// Mitsubishi GX Works2 project: zadatak_1_with_error   PLC: FX3S

// global labels: Global1
VAR_GLOBAL
  out_zone : zona_izlaza;
  fsm_1 : fsm;
  in_zone : zona_ulaza;
END_VAR

// task Task_01 (event TRUE, interval 0, priority 31): POU_01

PROGRAM POU_01
VAR
  system_on : BOOL;
  start : BOOL;
  stop_all : BOOL;
  start_all : BOOL;
  pump_on : BOOL;
  goto_1 : BOOL;
  goto_2 : BOOL;
  goto_3 : BOOL;
  goto_4 : BOOL;
  goto_0 : BOOL;
  cur_state : INT;
  s_0 : BOOL;
  s_1 : BOOL;
  s_2 : BOOL;
  s_3 : BOOL;
  s_4 : BOOL;
  sensor_2 : BOOL;
END_VAR
VAR CONSTANT
  pause : TIME := T#10s;
END_VAR
VAR
  elapsed_time : TIME;
  sensor_1 : BOOL;
  water_rising : BOOL;
  valve_1 : BOOL;
  motor : BOOL;
  water_falling : BOOL;
  valve_2 : BOOL;
  alarm : BOOL;
  TON_1 : TON;
  cnt_cycles_1 : cnt_cycles;
  done : BOOL;
  blink_1 : blink;
  lamp : BOOL;
  state : INT;
  enb : BOOL;
  sON : BOOL;
  zona_izlaz : zona_izlaza;
  zona_ulazz : zona_ulaza;
END_VAR
(* structured ladder/FBD written out as ST: instructions are called as NAME(EN, inputs, outputs); _pN, _eN, _tN stand for wires *)
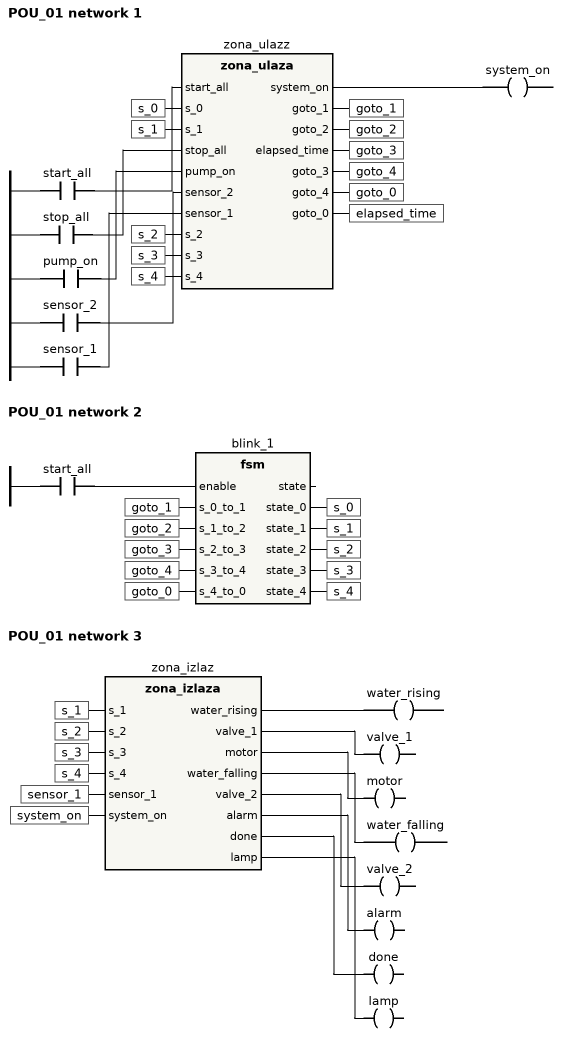
(* network 1 *)
zona_ulazz(start_all := start_all, s_0 := s_0, s_1 := s_1, stop_all := stop_all, pump_on := pump_on, sensor_2 := sensor_2, sensor_1 := sensor_1, s_2 := s_2, s_3 := s_3, s_4 := s_4, goto_1 => goto_1, goto_2 => goto_2, elapsed_time => goto_3, goto_3 => goto_4, goto_4 => goto_0, goto_0 => elapsed_time);
system_on := zona_ulazz.system_on;
(* network 2 *)
blink_1(enable := start_all, s_0_to_1 := goto_1, s_1_to_2 := goto_2, s_2_to_3 := goto_3, s_3_to_4 := goto_4, s_4_to_0 := goto_0, state_0 => s_0, state_1 => s_1, state_2 => s_2, state_3 => s_3, state_4 => s_4);
(* network 3 *)
zona_izlaz(s_1 := s_1, s_2 := s_2, s_3 := s_3, s_4 := s_4, sensor_1 := sensor_1, system_on := system_on);
water_rising := zona_izlaz.water_rising;
valve_1 := zona_izlaz.valve_1;
motor := zona_izlaz.motor;
water_falling := zona_izlaz.water_falling;
valve_2 := zona_izlaz.valve_2;
alarm := zona_izlaz.alarm;
done := zona_izlaz.done;
lamp := zona_izlaz.lamp;
END_PROGRAM

FUNCTION_BLOCK fsm
VAR_OUTPUT
  state : INT;
END_VAR
VAR CONSTANT
  cmp_with_0 : INT;
END_VAR
VAR
  is_eqv : ARRAY [0..2] OF BOOL;
END_VAR
VAR_INPUT
  enable : BOOL;
  s_0_to_1 : BOOL;
END_VAR
VAR_OUTPUT
  state_0 : BOOL;
END_VAR
VAR CONSTANT
  cmp_with_1 : INT := 1;
END_VAR
VAR_INPUT
  s_1_to_2 : BOOL;
END_VAR
VAR_OUTPUT
  state_1 : BOOL;
END_VAR
VAR CONSTANT
  cmp_with_2 : INT := 2;
END_VAR
VAR_INPUT
  s_2_to_3 : BOOL;
END_VAR
VAR_OUTPUT
  state_2 : BOOL;
  state_3 : BOOL;
END_VAR
VAR_INPUT
  s_3_to_4 : BOOL;
END_VAR
VAR CONSTANT
  cmp_with_4 : INT := 4;
  cmp_with_3 : INT := 3;
END_VAR
VAR_OUTPUT
  state_4 : BOOL;
END_VAR
VAR_INPUT
  s_4_to_0 : BOOL;
END_VAR
VAR
  blink_1 : blink;
END_VAR
(* structured ladder/FBD written out as ST: instructions are called as NAME(EN, inputs, outputs); _pN, _eN, _tN stand for wires *)
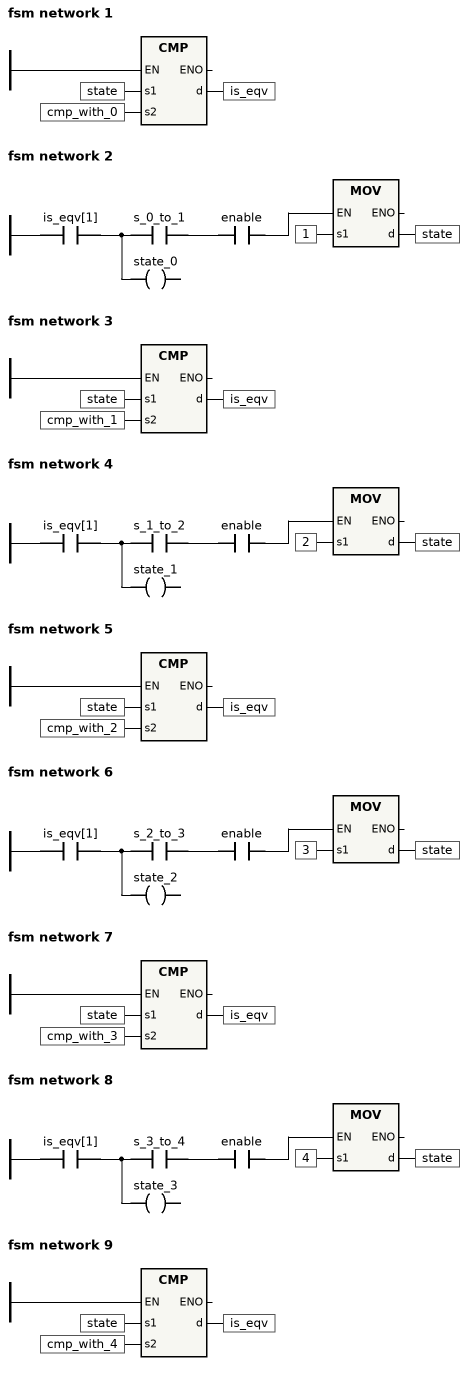
(* network 1 *)
CMP(TRUE, state, cmp_with_0, is_eqv);
(* network 2 *)
MOV(is_eqv[1] AND s_0_to_1 AND enable, 1, state);
state_0 := is_eqv[1];
(* network 3 *)
CMP(TRUE, state, cmp_with_1, is_eqv);
(* network 4 *)
MOV(is_eqv[1] AND s_1_to_2 AND enable, 2, state);
state_1 := is_eqv[1];
(* network 5 *)
CMP(TRUE, state, cmp_with_2, is_eqv);
(* network 6 *)
MOV(is_eqv[1] AND s_2_to_3 AND enable, 3, state);
state_2 := is_eqv[1];
(* network 7 *)
CMP(TRUE, state, cmp_with_3, is_eqv);
(* network 8 *)
MOV(is_eqv[1] AND s_3_to_4 AND enable, 4, state);
state_3 := is_eqv[1];
(* network 9 *)
CMP(TRUE, state, cmp_with_4, is_eqv);
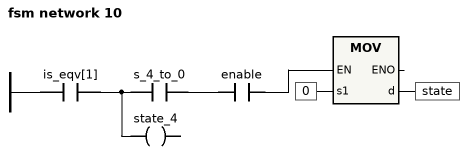
(* network 10 *)
MOV(is_eqv[1] AND s_4_to_0 AND enable, 0, state);
state_4 := is_eqv[1];
END_FUNCTION_BLOCK

FUNCTION_BLOCK cnt_cycles
VAR_INPUT
  cnt_start : BOOL;
END_VAR
VAR
  num_of_cycles : INT;
END_VAR
VAR CONSTANT
  add_1 : INT := 1;
END_VAR
VAR
  is_eqv : ARRAY [0..2] OF BOOL;
END_VAR
VAR CONSTANT
  cmp_with_5 : INT := 5;
END_VAR
VAR_OUTPUT
  done : BOOL;
END_VAR
(* structured ladder/FBD written out as ST: instructions are called as NAME(EN, inputs, outputs); _pN, _eN, _tN stand for wires *)
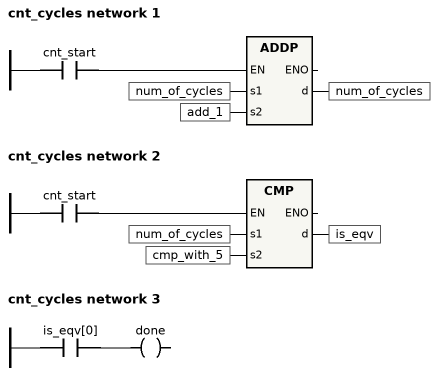
(* network 1 *)
ADDP(cnt_start, num_of_cycles, add_1, num_of_cycles);
(* network 2 *)
CMP(cnt_start, num_of_cycles, cmp_with_5, is_eqv);
(* network 3 *)
done := is_eqv[0];
END_FUNCTION_BLOCK

FUNCTION_BLOCK blink
VAR_INPUT
  ulaz : BOOL;
END_VAR
VAR_OUTPUT
  radi : BOOL;
END_VAR
VAR
  TON_1 : TON;
  TON_2 : TON;
  Tajmer1_izlaz : BOOL;
  Tajmer2_izlaz : BOOL;
  vreme_ton1 : TIME;
  vreme_ton2 : TIME;
END_VAR
IF ulaz=TRUE THEN
	
	TON_1(IN:=NOT Tajmer2_izlaz,PT:= T#1000ms,Q:=Tajmer1_izlaz,ET:=vreme_ton1);
	TON_2(IN:=NOT Tajmer2_izlaz,PT:= T#2000ms,Q:=Tajmer2_izlaz,ET:=vreme_ton2);
	
END_IF;

IF Tajmer1_izlaz=TRUE THEN radi:=TRUE;ELSE radi:=FALSE;
END_IF;
END_FUNCTION_BLOCK

FUNCTION_BLOCK zona_ulaza
VAR_INPUT
  start_all : BOOL;
  s_0 : BOOL;
  s_1 : BOOL;
  stop_all : BOOL;
  pump_on : BOOL;
  sensor_2 : BOOL;
  sensor_1 : BOOL;
  s_2 : BOOL;
  s_3 : BOOL;
  s_4 : BOOL;
END_VAR
VAR_OUTPUT
  system_on : BOOL;
  goto_1 : BOOL;
  goto_2 : BOOL;
  elapsed_time : TIME;
  goto_3 : BOOL;
  goto_4 : BOOL;
  goto_0 : BOOL;
END_VAR
VAR
  TON_1 : TON;
END_VAR
VAR CONSTANT
  pause : TIME := T#10s;
END_VAR
(* structured ladder/FBD written out as ST: instructions are called as NAME(EN, inputs, outputs); _pN, _eN, _tN stand for wires *)
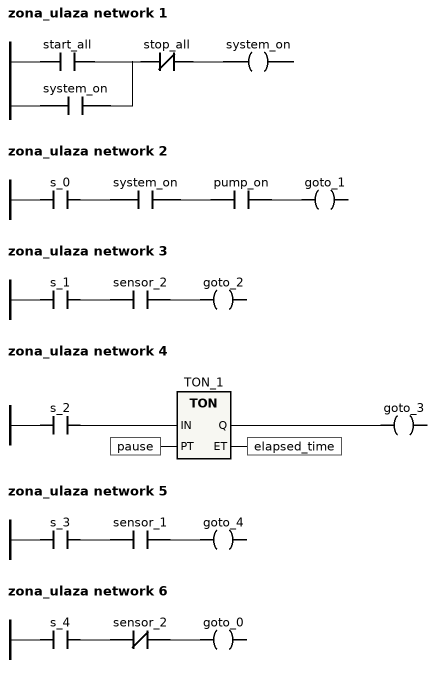
(* network 1 *)
system_on := (start_all OR system_on) AND NOT stop_all;
(* network 2 *)
goto_1 := s_0 AND system_on AND pump_on;
(* network 3 *)
goto_2 := s_1 AND sensor_2;
(* network 4 *)
TON_1(IN := s_2, PT := pause, ET => elapsed_time);
goto_3 := TON_1.Q;
(* network 5 *)
goto_4 := s_3 AND sensor_1;
(* network 6 *)
goto_0 := s_4 AND NOT sensor_2;
END_FUNCTION_BLOCK

FUNCTION_BLOCK zona_izlaza
VAR_INPUT
  s_1 : BOOL;
END_VAR
VAR_OUTPUT
  water_rising : BOOL;
  valve_1 : BOOL;
  motor : BOOL;
  water_falling : BOOL;
  valve_2 : BOOL;
  alarm : BOOL;
  done : BOOL;
  lamp : BOOL;
END_VAR
VAR_INPUT
  s_2 : BOOL;
  s_3 : BOOL;
  s_4 : BOOL;
  sensor_1 : BOOL;
  system_on : BOOL;
END_VAR
VAR
  cnt_cycles_1 : cnt_cycles;
  blink_1 : blink;
END_VAR
(* structured ladder/FBD written out as ST: instructions are called as NAME(EN, inputs, outputs); _pN, _eN, _tN stand for wires *)
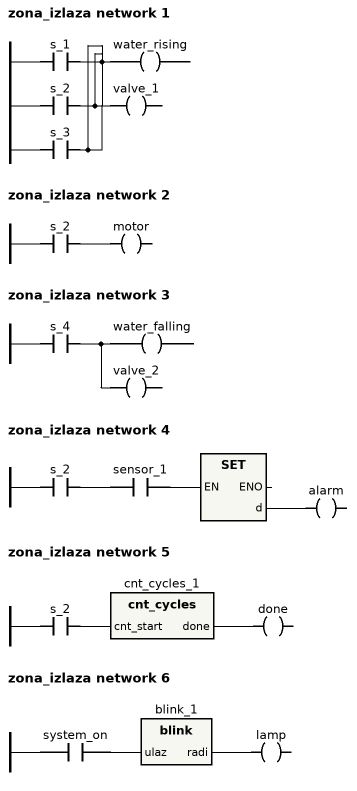
(* network 1 *)
_p1 := s_1 OR s_2 OR s_3;
water_rising := _p1;
valve_1 := _p1;
(* network 2 *)
motor := s_2;
(* network 3 *)
water_falling := s_4;
valve_2 := s_4;
(* network 4 *)
SET(s_2 AND sensor_1, _t1);
alarm := _t1;
(* network 5 *)
cnt_cycles_1(cnt_start := s_2);
done := cnt_cycles_1.done;
(* network 6 *)
blink_1(ulaz := system_on);
lamp := blink_1.radi;
END_FUNCTION_BLOCK
